TYPE stRelativePose3D :
STRUCT
    dx : LREAL;
    dy : LREAL;
    dz : LREAL;
    drx : LREAL;
    dry : LREAL;
    drz : LREAL;
END_STRUCT
END_TYPE

(* stored: Version 1.1.0.1, ProductVersion 3.1.4026.18
   DUT stRelativePose3D: Id {6e85a8f2-cc8a-4c4a-9c20-4e5dfbd91148} *)
